// TIA Portal V17 export
// export: Created 2025-03-05T08:01:40.0178288Z, ExportSetting WithDefaults, DisplayName Totally Integrated Automation Portal, DisplayVersion V17 Update 8, DisplayName TIA Portal Openness, DisplayVersion V17 Update 8, DisplayName TIA Portal Version Control Interface, DisplayVersion V17, DisplayName SINAMICS Startdrive Advanced, DisplayVersion V17 SP2, DisplayName SINAMICS Startdrive G110M, G120, G120C, G120D, G120P, G115D, DisplayVersion V17 SP2, DisplayName SINAMICS Startdrive G130, G150, S120, S150, SINAMICS MV, S210, DisplayVersion V17 SP2, DisplayName STEP 7 Professional, DisplayVersion V17 Update 8, DisplayName SINUMERIK ONE STEP 7 Toolbox, DisplayVersion V17 Update 12, DisplayName SINUMERIK 840D sl STEP 7 Toolbox, DisplayVersion V17 Update 12, DisplayName STEP 7 Safety, DisplayVersion V17 Update 6, DisplayName WinCC Advanced, DisplayVersion V17 Update 8
FUNCTION "FC7215_PART_TYPE" : Void   // FC7215, LAD
{ S7_Optimized_Access := 'FALSE' }
AUTHOR : ETXETAR
VERSION : 1.0
// stored: AutoNumber false, IsIECCheckEnabled false, SetENOAutomatically false, UDAEnableTagReadback false
   VAR_TEMP
      PART_TYPE_SCREEN : Int;   // PART TYPE SCREEN
   END_VAR
   VAR CONSTANT
      FC_NUMBER : DInt := 7215;
   END_VAR
   VAR_TEMP   // added for the SCL form of the ladder/FBD networks
      _w1 : Bool;
      _w2 : Bool;
   END_VAR
BEGIN

REGION Network 1: AUTO PART TYPE SELECT
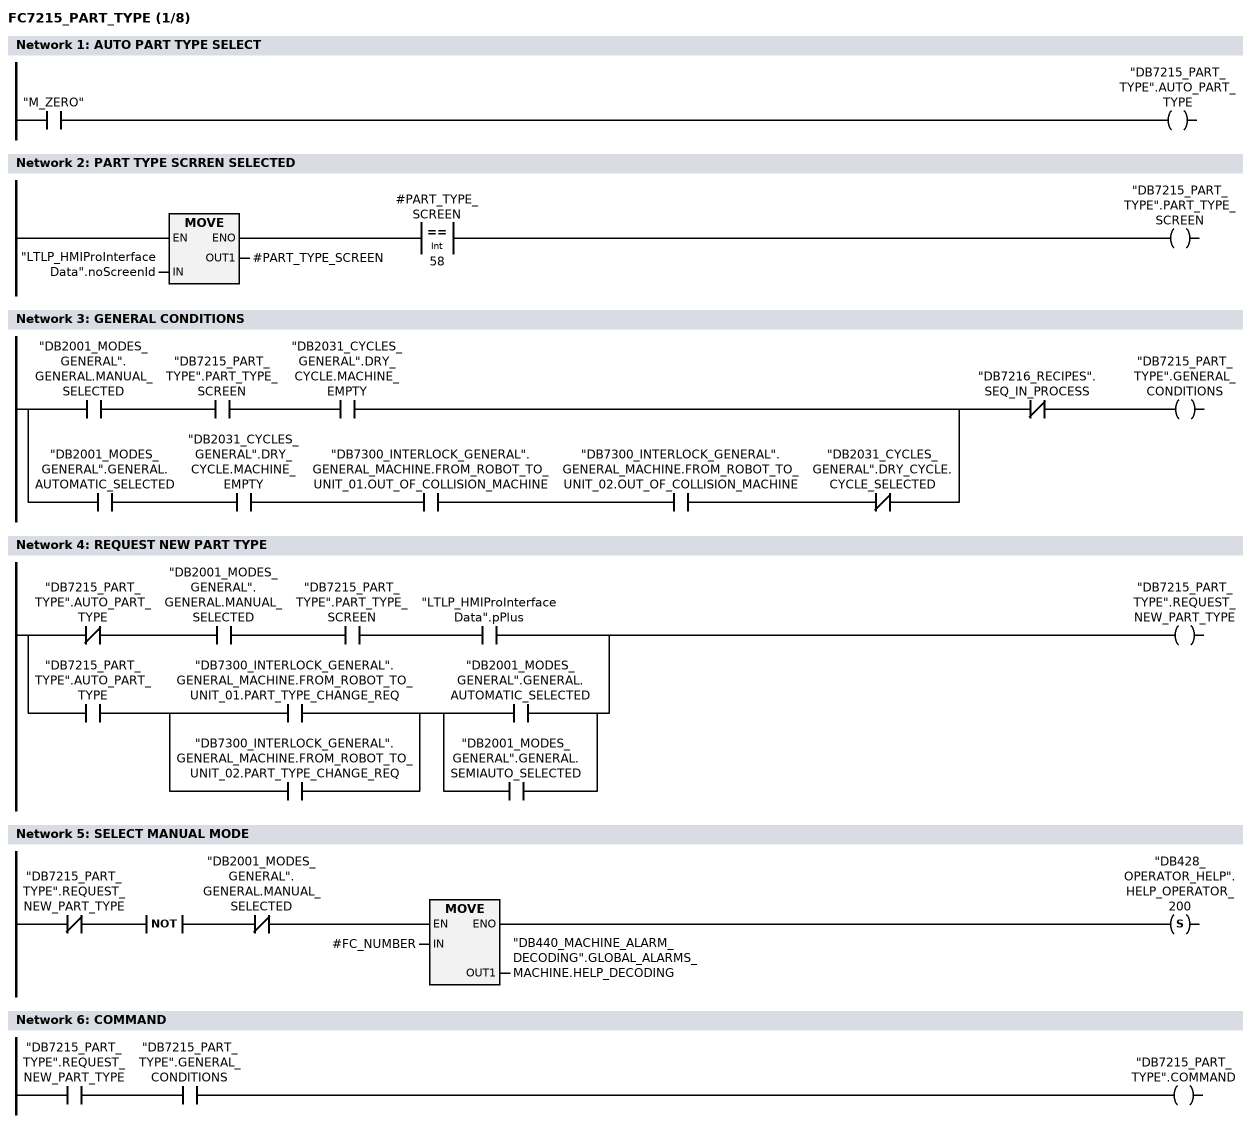
   RUNG wire#powerrail
      Contact( "M_ZERO" )
      Coil( "DB7215_PART_TYPE".AUTO_PART_TYPE )
   END_RUNG
   // the same network as SCL:
   "DB7215_PART_TYPE".AUTO_PART_TYPE := "M_ZERO";
END_REGION

REGION Network 2: PART TYPE SCRREN SELECTED
   RUNG wire#powerrail
      { S7_GenerateENO := "TRUE" } Move(in := "LTLP_HMIProInterfaceData".noScreenId, out1 => #PART_TYPE_SCREEN)
      { S7_Templates := "SrcType := Int" } EQ_Contact(in1 := #PART_TYPE_SCREEN, in2 := 58)
      Coil( "DB7215_PART_TYPE".PART_TYPE_SCREEN )
   END_RUNG
   // the same network as SCL:
   // ENO of a box is taken as its EN; it also drops when the box reports an error
   #PART_TYPE_SCREEN := "LTLP_HMIProInterfaceData".noScreenId;
   "DB7215_PART_TYPE".PART_TYPE_SCREEN := #PART_TYPE_SCREEN = 58;
END_REGION

REGION Network 3: GENERAL CONDITIONS
   RUNG wire#powerrail
      Contact( "DB2001_MODES_GENERAL".GENERAL.MANUAL_SELECTED )
      Contact( "DB7215_PART_TYPE".PART_TYPE_SCREEN )
      Contact( "DB2031_CYCLES_GENERAL".DRY_CYCLE.MACHINE_EMPTY )
      wire#w1
      I_Contact( "DB7216_RECIPES".SEQ_IN_PROCESS )
      Coil( "DB7215_PART_TYPE".GENERAL_CONDITIONS )
   END_RUNG
   RUNG wire#powerrail
      Contact( "DB2001_MODES_GENERAL".GENERAL.AUTOMATIC_SELECTED )
      Contact( "DB2031_CYCLES_GENERAL".DRY_CYCLE.MACHINE_EMPTY )
      Contact( "DB7300_INTERLOCK_GENERAL".GENERAL_MACHINE.FROM_ROBOT_TO_UNIT_01.OUT_OF_COLLISION_MACHINE )
      Contact( "DB7300_INTERLOCK_GENERAL".GENERAL_MACHINE.FROM_ROBOT_TO_UNIT_02.OUT_OF_COLLISION_MACHINE )
      I_Contact( "DB2031_CYCLES_GENERAL".DRY_CYCLE.CYCLE_SELECTED )
   END_RUNG wire#w1
   // the same network as SCL:
   "DB7215_PART_TYPE".GENERAL_CONDITIONS := (("DB2001_MODES_GENERAL".GENERAL.MANUAL_SELECTED AND "DB7215_PART_TYPE".PART_TYPE_SCREEN AND "DB2031_CYCLES_GENERAL".DRY_CYCLE.MACHINE_EMPTY) OR ("DB2001_MODES_GENERAL".GENERAL.AUTOMATIC_SELECTED AND "DB2031_CYCLES_GENERAL".DRY_CYCLE.MACHINE_EMPTY AND "DB7300_INTERLOCK_GENERAL".GENERAL_MACHINE.FROM_ROBOT_TO_UNIT_01.OUT_OF_COLLISION_MACHINE AND "DB7300_INTERLOCK_GENERAL".GENERAL_MACHINE.FROM_ROBOT_TO_UNIT_02.OUT_OF_COLLISION_MACHINE AND NOT "DB2031_CYCLES_GENERAL".DRY_CYCLE.CYCLE_SELECTED)) AND NOT "DB7216_RECIPES".SEQ_IN_PROCESS;
END_REGION

REGION Network 4: REQUEST NEW PART TYPE
   RUNG wire#powerrail
      I_Contact( "DB7215_PART_TYPE".AUTO_PART_TYPE )
      Contact( "DB2001_MODES_GENERAL".GENERAL.MANUAL_SELECTED )
      Contact( "DB7215_PART_TYPE".PART_TYPE_SCREEN )
      Contact( "LTLP_HMIProInterfaceData".pPlus )
      wire#w1
      Coil( "DB7215_PART_TYPE".REQUEST_NEW_PART_TYPE )
   END_RUNG
   RUNG wire#powerrail
      Contact( "DB7215_PART_TYPE".AUTO_PART_TYPE )
      wire#w2
      Contact( "DB7300_INTERLOCK_GENERAL".GENERAL_MACHINE.FROM_ROBOT_TO_UNIT_01.PART_TYPE_CHANGE_REQ )
      wire#w3
      Contact( "DB2001_MODES_GENERAL".GENERAL.AUTOMATIC_SELECTED )
   END_RUNG wire#w1
   RUNG wire#w2
      Contact( "DB7300_INTERLOCK_GENERAL".GENERAL_MACHINE.FROM_ROBOT_TO_UNIT_02.PART_TYPE_CHANGE_REQ )
   END_RUNG wire#w3
   RUNG wire#w3
      Contact( "DB2001_MODES_GENERAL".GENERAL.SEMIAUTO_SELECTED )
   END_RUNG wire#w1
   // the same network as SCL:
   "DB7215_PART_TYPE".REQUEST_NEW_PART_TYPE := (NOT "DB7215_PART_TYPE".AUTO_PART_TYPE AND "DB2001_MODES_GENERAL".GENERAL.MANUAL_SELECTED AND "DB7215_PART_TYPE".PART_TYPE_SCREEN AND "LTLP_HMIProInterfaceData".pPlus) OR ("DB7215_PART_TYPE".AUTO_PART_TYPE AND ("DB7300_INTERLOCK_GENERAL".GENERAL_MACHINE.FROM_ROBOT_TO_UNIT_01.PART_TYPE_CHANGE_REQ OR "DB7300_INTERLOCK_GENERAL".GENERAL_MACHINE.FROM_ROBOT_TO_UNIT_02.PART_TYPE_CHANGE_REQ) AND ("DB2001_MODES_GENERAL".GENERAL.AUTOMATIC_SELECTED OR "DB2001_MODES_GENERAL".GENERAL.SEMIAUTO_SELECTED));
END_REGION

REGION Network 5: SELECT MANUAL MODE
   RUNG wire#powerrail
      I_Contact( "DB7215_PART_TYPE".REQUEST_NEW_PART_TYPE )
      Not()
      I_Contact( "DB2001_MODES_GENERAL".GENERAL.MANUAL_SELECTED )
      { S7_GenerateENO := "TRUE" } Move(in := #FC_NUMBER, out1 => "DB440_MACHINE_ALARM_DECODING".GLOBAL_ALARMS_MACHINE.HELP_DECODING)
      S_Coil( "DB428_OPERATOR_HELP".HELP_OPERATOR_200 )
   END_RUNG
   // the same network as SCL:
   // ENO of a box is taken as its EN; it also drops when the box reports an error
   IF NOT (NOT "DB7215_PART_TYPE".REQUEST_NEW_PART_TYPE) AND NOT "DB2001_MODES_GENERAL".GENERAL.MANUAL_SELECTED THEN
       "DB440_MACHINE_ALARM_DECODING".GLOBAL_ALARMS_MACHINE.HELP_DECODING := #FC_NUMBER;
       "DB428_OPERATOR_HELP".HELP_OPERATOR_200 := TRUE;
   END_IF;
END_REGION

REGION Network 6: COMMAND
   RUNG wire#powerrail
      Contact( "DB7215_PART_TYPE".REQUEST_NEW_PART_TYPE )
      Contact( "DB7215_PART_TYPE".GENERAL_CONDITIONS )
      Coil( "DB7215_PART_TYPE".COMMAND )
   END_RUNG
   // the same network as SCL:
   "DB7215_PART_TYPE".COMMAND := "DB7215_PART_TYPE".REQUEST_NEW_PART_TYPE AND "DB7215_PART_TYPE".GENERAL_CONDITIONS;
END_REGION

REGION Network 7: COMMAND
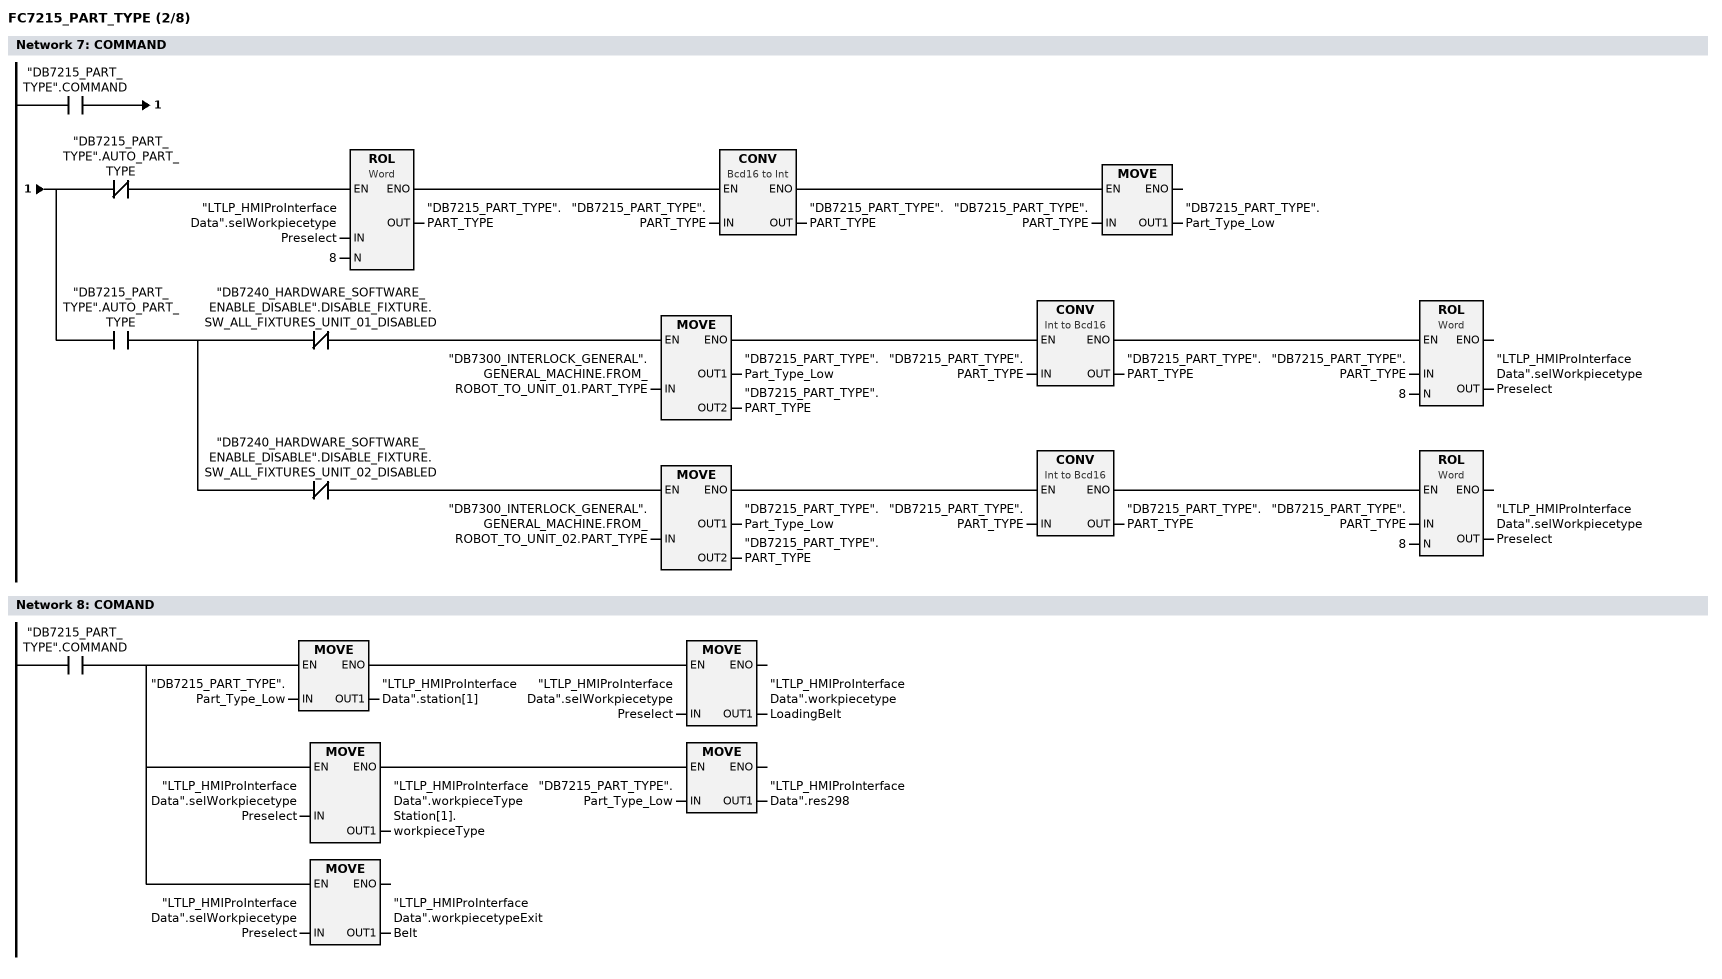
   IF "DB7215_PART_TYPE".COMMAND AND NOT "DB7215_PART_TYPE".AUTO_PART_TYPE THEN
       "DB7215_PART_TYPE".PART_TYPE := ROL(IN := "LTLP_HMIProInterfaceData".selWorkpiecetypePreselect, N := 8);
       "DB7215_PART_TYPE".PART_TYPE := BCD16_TO_INT("DB7215_PART_TYPE".PART_TYPE);
       "DB7215_PART_TYPE".Part_Type_Low := "DB7215_PART_TYPE".PART_TYPE;
   END_IF;
   #_w1 := "DB7215_PART_TYPE".COMMAND AND "DB7215_PART_TYPE".AUTO_PART_TYPE;
   IF #_w1 AND NOT "DB7240_HARDWARE_SOFTWARE_ENABLE_DISABLE".DISABLE_FIXTURE.SW_ALL_FIXTURES_UNIT_01_DISABLED THEN
       "DB7215_PART_TYPE".Part_Type_Low := "DB7300_INTERLOCK_GENERAL".GENERAL_MACHINE.FROM_ROBOT_TO_UNIT_01.PART_TYPE;
       "DB7215_PART_TYPE".PART_TYPE := "DB7300_INTERLOCK_GENERAL".GENERAL_MACHINE.FROM_ROBOT_TO_UNIT_01.PART_TYPE;
       "DB7215_PART_TYPE".PART_TYPE := INT_TO_BCD16("DB7215_PART_TYPE".PART_TYPE);
       "LTLP_HMIProInterfaceData".selWorkpiecetypePreselect := ROL(IN := "DB7215_PART_TYPE".PART_TYPE, N := 8);
   END_IF;
   IF #_w1 AND NOT "DB7240_HARDWARE_SOFTWARE_ENABLE_DISABLE".DISABLE_FIXTURE.SW_ALL_FIXTURES_UNIT_02_DISABLED THEN
       "DB7215_PART_TYPE".Part_Type_Low := "DB7300_INTERLOCK_GENERAL".GENERAL_MACHINE.FROM_ROBOT_TO_UNIT_02.PART_TYPE;
       "DB7215_PART_TYPE".PART_TYPE := "DB7300_INTERLOCK_GENERAL".GENERAL_MACHINE.FROM_ROBOT_TO_UNIT_02.PART_TYPE;
       "DB7215_PART_TYPE".PART_TYPE := INT_TO_BCD16("DB7215_PART_TYPE".PART_TYPE);
       "LTLP_HMIProInterfaceData".selWorkpiecetypePreselect := ROL(IN := "DB7215_PART_TYPE".PART_TYPE, N := 8);
   END_IF;
END_REGION

REGION Network 8: COMAND
   RUNG wire#powerrail
      Contact( "DB7215_PART_TYPE".COMMAND )
      wire#w1
      { S7_GenerateENO := "TRUE" } Move(in := "DB7215_PART_TYPE".Part_Type_Low, out1 => "LTLP_HMIProInterfaceData".station[1])
      { S7_GenerateENO := "TRUE" } Move(in := "LTLP_HMIProInterfaceData".selWorkpiecetypePreselect, out1 => "LTLP_HMIProInterfaceData".workpiecetypeLoadingBelt)
   END_RUNG
   RUNG wire#w1
      { S7_GenerateENO := "TRUE" } Move(in := "LTLP_HMIProInterfaceData".selWorkpiecetypePreselect, out1 => "LTLP_HMIProInterfaceData".workpieceTypeStation[1].workpieceType)
      { S7_GenerateENO := "TRUE" } Move(in := "DB7215_PART_TYPE".Part_Type_Low, out1 => "LTLP_HMIProInterfaceData".res298)
   END_RUNG
   RUNG wire#w1
      { S7_GenerateENO := "TRUE" } Move(in := "LTLP_HMIProInterfaceData".selWorkpiecetypePreselect, out1 => "LTLP_HMIProInterfaceData".workpiecetypeExitBelt)
   END_RUNG
   // the same network as SCL:
   // ENO of a box is taken as its EN; it also drops when the box reports an error
   IF "DB7215_PART_TYPE".COMMAND THEN
       "LTLP_HMIProInterfaceData".station[1] := "DB7215_PART_TYPE".Part_Type_Low;
       "LTLP_HMIProInterfaceData".workpiecetypeLoadingBelt := "LTLP_HMIProInterfaceData".selWorkpiecetypePreselect;
       "LTLP_HMIProInterfaceData".workpieceTypeStation[1].workpieceType := "LTLP_HMIProInterfaceData".selWorkpiecetypePreselect;
       "LTLP_HMIProInterfaceData".res298 := "DB7215_PART_TYPE".Part_Type_Low;
       "LTLP_HMIProInterfaceData".workpiecetypeExitBelt := "LTLP_HMIProInterfaceData".selWorkpiecetypePreselect;
   END_IF;
END_REGION

REGION Network 9: PART TYPE SELECTED 1 - 8
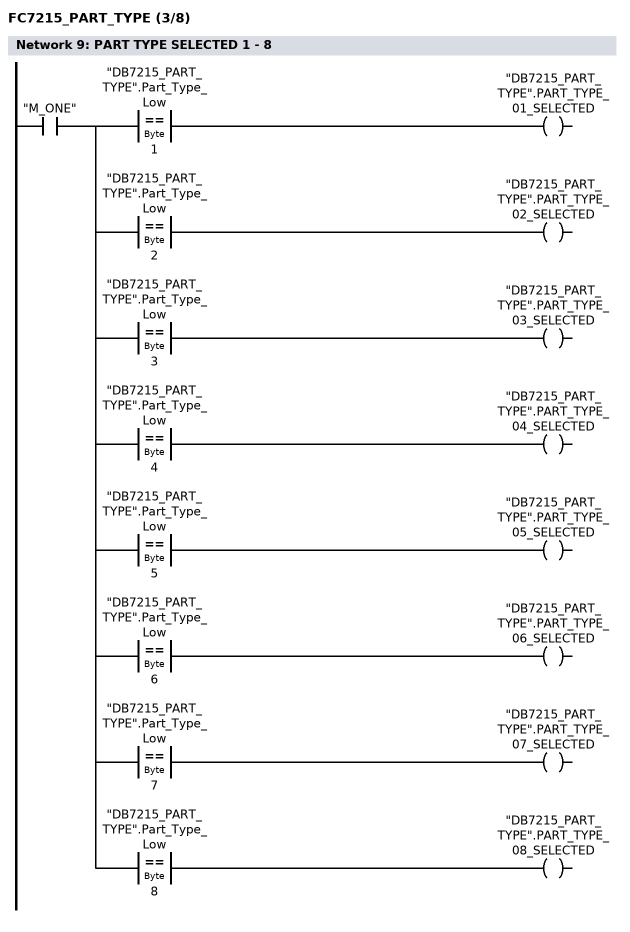
   RUNG wire#powerrail
      Contact( "M_ONE" )
      wire#w1
      { S7_Templates := "SrcType := Byte" } EQ_Contact(in1 := "DB7215_PART_TYPE".Part_Type_Low, in2 := 1)
      Coil( "DB7215_PART_TYPE".PART_TYPE_01_SELECTED )
   END_RUNG
   RUNG wire#w1
      { S7_Templates := "SrcType := Byte" } EQ_Contact(in1 := "DB7215_PART_TYPE".Part_Type_Low, in2 := 2)
      Coil( "DB7215_PART_TYPE".PART_TYPE_02_SELECTED )
   END_RUNG
   RUNG wire#w1
      { S7_Templates := "SrcType := Byte" } EQ_Contact(in1 := "DB7215_PART_TYPE".Part_Type_Low, in2 := 3)
      Coil( "DB7215_PART_TYPE".PART_TYPE_03_SELECTED )
   END_RUNG
   RUNG wire#w1
      { S7_Templates := "SrcType := Byte" } EQ_Contact(in1 := "DB7215_PART_TYPE".Part_Type_Low, in2 := 4)
      Coil( "DB7215_PART_TYPE".PART_TYPE_04_SELECTED )
   END_RUNG
   RUNG wire#w1
      { S7_Templates := "SrcType := Byte" } EQ_Contact(in1 := "DB7215_PART_TYPE".Part_Type_Low, in2 := 5)
      Coil( "DB7215_PART_TYPE".PART_TYPE_05_SELECTED )
   END_RUNG
   RUNG wire#w1
      { S7_Templates := "SrcType := Byte" } EQ_Contact(in1 := "DB7215_PART_TYPE".Part_Type_Low, in2 := 6)
      Coil( "DB7215_PART_TYPE".PART_TYPE_06_SELECTED )
   END_RUNG
   RUNG wire#w1
      { S7_Templates := "SrcType := Byte" } EQ_Contact(in1 := "DB7215_PART_TYPE".Part_Type_Low, in2 := 7)
      Coil( "DB7215_PART_TYPE".PART_TYPE_07_SELECTED )
   END_RUNG
   RUNG wire#w1
      { S7_Templates := "SrcType := Byte" } EQ_Contact(in1 := "DB7215_PART_TYPE".Part_Type_Low, in2 := 8)
      Coil( "DB7215_PART_TYPE".PART_TYPE_08_SELECTED )
   END_RUNG
   // the same network as SCL:
   "DB7215_PART_TYPE".PART_TYPE_01_SELECTED := "M_ONE" AND ("DB7215_PART_TYPE".Part_Type_Low = 1);
   "DB7215_PART_TYPE".PART_TYPE_02_SELECTED := "M_ONE" AND ("DB7215_PART_TYPE".Part_Type_Low = 2);
   "DB7215_PART_TYPE".PART_TYPE_03_SELECTED := "M_ONE" AND ("DB7215_PART_TYPE".Part_Type_Low = 3);
   "DB7215_PART_TYPE".PART_TYPE_04_SELECTED := "M_ONE" AND ("DB7215_PART_TYPE".Part_Type_Low = 4);
   "DB7215_PART_TYPE".PART_TYPE_05_SELECTED := "M_ONE" AND ("DB7215_PART_TYPE".Part_Type_Low = 5);
   "DB7215_PART_TYPE".PART_TYPE_06_SELECTED := "M_ONE" AND ("DB7215_PART_TYPE".Part_Type_Low = 6);
   "DB7215_PART_TYPE".PART_TYPE_07_SELECTED := "M_ONE" AND ("DB7215_PART_TYPE".Part_Type_Low = 7);
   "DB7215_PART_TYPE".PART_TYPE_08_SELECTED := "M_ONE" AND ("DB7215_PART_TYPE".Part_Type_Low = 8);
END_REGION

REGION Network 10: PART TYPE SELECTED 9 - 16
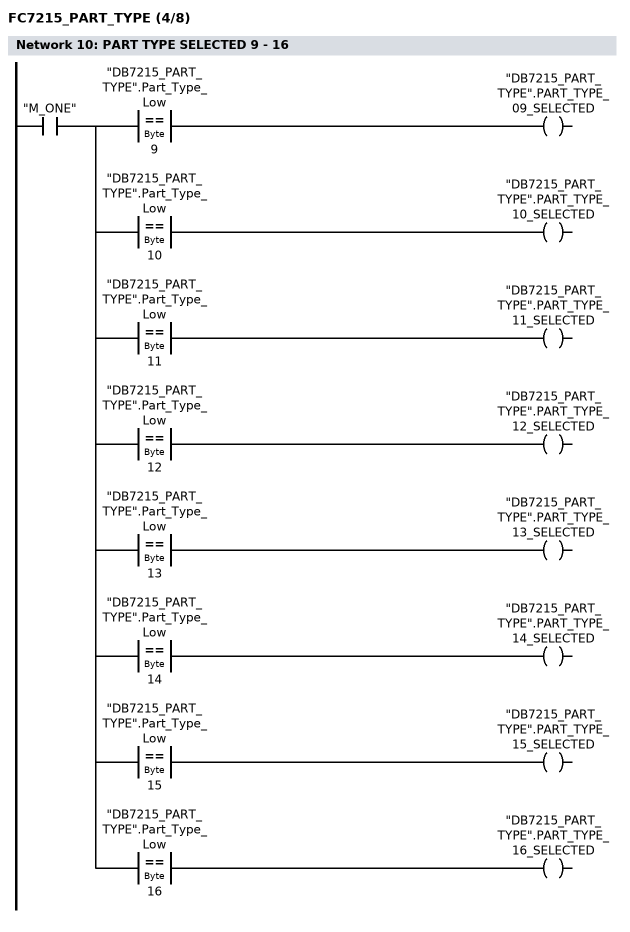
   RUNG wire#powerrail
      Contact( "M_ONE" )
      wire#w1
      { S7_Templates := "SrcType := Byte" } EQ_Contact(in1 := "DB7215_PART_TYPE".Part_Type_Low, in2 := 9)
      Coil( "DB7215_PART_TYPE".PART_TYPE_09_SELECTED )
   END_RUNG
   RUNG wire#w1
      { S7_Templates := "SrcType := Byte" } EQ_Contact(in1 := "DB7215_PART_TYPE".Part_Type_Low, in2 := 10)
      Coil( "DB7215_PART_TYPE".PART_TYPE_10_SELECTED )
   END_RUNG
   RUNG wire#w1
      { S7_Templates := "SrcType := Byte" } EQ_Contact(in1 := "DB7215_PART_TYPE".Part_Type_Low, in2 := 11)
      Coil( "DB7215_PART_TYPE".PART_TYPE_11_SELECTED )
   END_RUNG
   RUNG wire#w1
      { S7_Templates := "SrcType := Byte" } EQ_Contact(in1 := "DB7215_PART_TYPE".Part_Type_Low, in2 := 12)
      Coil( "DB7215_PART_TYPE".PART_TYPE_12_SELECTED )
   END_RUNG
   RUNG wire#w1
      { S7_Templates := "SrcType := Byte" } EQ_Contact(in1 := "DB7215_PART_TYPE".Part_Type_Low, in2 := 13)
      Coil( "DB7215_PART_TYPE".PART_TYPE_13_SELECTED )
   END_RUNG
   RUNG wire#w1
      { S7_Templates := "SrcType := Byte" } EQ_Contact(in1 := "DB7215_PART_TYPE".Part_Type_Low, in2 := 14)
      Coil( "DB7215_PART_TYPE".PART_TYPE_14_SELECTED )
   END_RUNG
   RUNG wire#w1
      { S7_Templates := "SrcType := Byte" } EQ_Contact(in1 := "DB7215_PART_TYPE".Part_Type_Low, in2 := 15)
      Coil( "DB7215_PART_TYPE".PART_TYPE_15_SELECTED )
   END_RUNG
   RUNG wire#w1
      { S7_Templates := "SrcType := Byte" } EQ_Contact(in1 := "DB7215_PART_TYPE".Part_Type_Low, in2 := 16)
      Coil( "DB7215_PART_TYPE".PART_TYPE_16_SELECTED )
   END_RUNG
   // the same network as SCL:
   "DB7215_PART_TYPE".PART_TYPE_09_SELECTED := "M_ONE" AND ("DB7215_PART_TYPE".Part_Type_Low = 9);
   "DB7215_PART_TYPE".PART_TYPE_10_SELECTED := "M_ONE" AND ("DB7215_PART_TYPE".Part_Type_Low = 10);
   "DB7215_PART_TYPE".PART_TYPE_11_SELECTED := "M_ONE" AND ("DB7215_PART_TYPE".Part_Type_Low = 11);
   "DB7215_PART_TYPE".PART_TYPE_12_SELECTED := "M_ONE" AND ("DB7215_PART_TYPE".Part_Type_Low = 12);
   "DB7215_PART_TYPE".PART_TYPE_13_SELECTED := "M_ONE" AND ("DB7215_PART_TYPE".Part_Type_Low = 13);
   "DB7215_PART_TYPE".PART_TYPE_14_SELECTED := "M_ONE" AND ("DB7215_PART_TYPE".Part_Type_Low = 14);
   "DB7215_PART_TYPE".PART_TYPE_15_SELECTED := "M_ONE" AND ("DB7215_PART_TYPE".Part_Type_Low = 15);
   "DB7215_PART_TYPE".PART_TYPE_16_SELECTED := "M_ONE" AND ("DB7215_PART_TYPE".Part_Type_Low = 16);
END_REGION

REGION Network 11: PART TYPE SELECTED 17 - 24
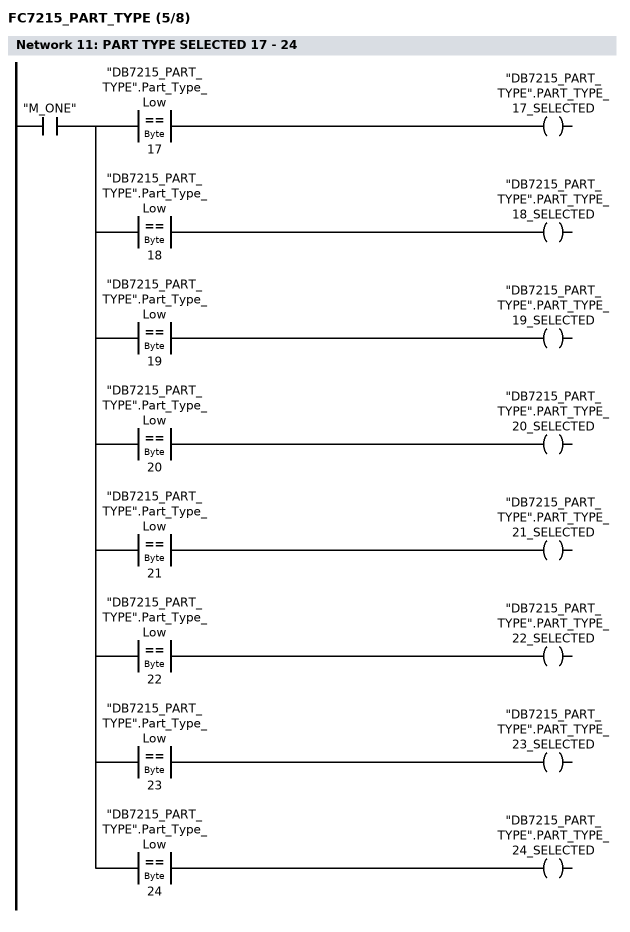
   RUNG wire#powerrail
      Contact( "M_ONE" )
      wire#w1
      { S7_Templates := "SrcType := Byte" } EQ_Contact(in1 := "DB7215_PART_TYPE".Part_Type_Low, in2 := 17)
      Coil( "DB7215_PART_TYPE".PART_TYPE_17_SELECTED )
   END_RUNG
   RUNG wire#w1
      { S7_Templates := "SrcType := Byte" } EQ_Contact(in1 := "DB7215_PART_TYPE".Part_Type_Low, in2 := 18)
      Coil( "DB7215_PART_TYPE".PART_TYPE_18_SELECTED )
   END_RUNG
   RUNG wire#w1
      { S7_Templates := "SrcType := Byte" } EQ_Contact(in1 := "DB7215_PART_TYPE".Part_Type_Low, in2 := 19)
      Coil( "DB7215_PART_TYPE".PART_TYPE_19_SELECTED )
   END_RUNG
   RUNG wire#w1
      { S7_Templates := "SrcType := Byte" } EQ_Contact(in1 := "DB7215_PART_TYPE".Part_Type_Low, in2 := 20)
      Coil( "DB7215_PART_TYPE".PART_TYPE_20_SELECTED )
   END_RUNG
   RUNG wire#w1
      { S7_Templates := "SrcType := Byte" } EQ_Contact(in1 := "DB7215_PART_TYPE".Part_Type_Low, in2 := 21)
      Coil( "DB7215_PART_TYPE".PART_TYPE_21_SELECTED )
   END_RUNG
   RUNG wire#w1
      { S7_Templates := "SrcType := Byte" } EQ_Contact(in1 := "DB7215_PART_TYPE".Part_Type_Low, in2 := 22)
      Coil( "DB7215_PART_TYPE".PART_TYPE_22_SELECTED )
   END_RUNG
   RUNG wire#w1
      { S7_Templates := "SrcType := Byte" } EQ_Contact(in1 := "DB7215_PART_TYPE".Part_Type_Low, in2 := 23)
      Coil( "DB7215_PART_TYPE".PART_TYPE_23_SELECTED )
   END_RUNG
   RUNG wire#w1
      { S7_Templates := "SrcType := Byte" } EQ_Contact(in1 := "DB7215_PART_TYPE".Part_Type_Low, in2 := 24)
      Coil( "DB7215_PART_TYPE".PART_TYPE_24_SELECTED )
   END_RUNG
   // the same network as SCL:
   "DB7215_PART_TYPE".PART_TYPE_17_SELECTED := "M_ONE" AND ("DB7215_PART_TYPE".Part_Type_Low = 17);
   "DB7215_PART_TYPE".PART_TYPE_18_SELECTED := "M_ONE" AND ("DB7215_PART_TYPE".Part_Type_Low = 18);
   "DB7215_PART_TYPE".PART_TYPE_19_SELECTED := "M_ONE" AND ("DB7215_PART_TYPE".Part_Type_Low = 19);
   "DB7215_PART_TYPE".PART_TYPE_20_SELECTED := "M_ONE" AND ("DB7215_PART_TYPE".Part_Type_Low = 20);
   "DB7215_PART_TYPE".PART_TYPE_21_SELECTED := "M_ONE" AND ("DB7215_PART_TYPE".Part_Type_Low = 21);
   "DB7215_PART_TYPE".PART_TYPE_22_SELECTED := "M_ONE" AND ("DB7215_PART_TYPE".Part_Type_Low = 22);
   "DB7215_PART_TYPE".PART_TYPE_23_SELECTED := "M_ONE" AND ("DB7215_PART_TYPE".Part_Type_Low = 23);
   "DB7215_PART_TYPE".PART_TYPE_24_SELECTED := "M_ONE" AND ("DB7215_PART_TYPE".Part_Type_Low = 24);
END_REGION

REGION Network 12: PART TYPE SELECTED 25 - 32
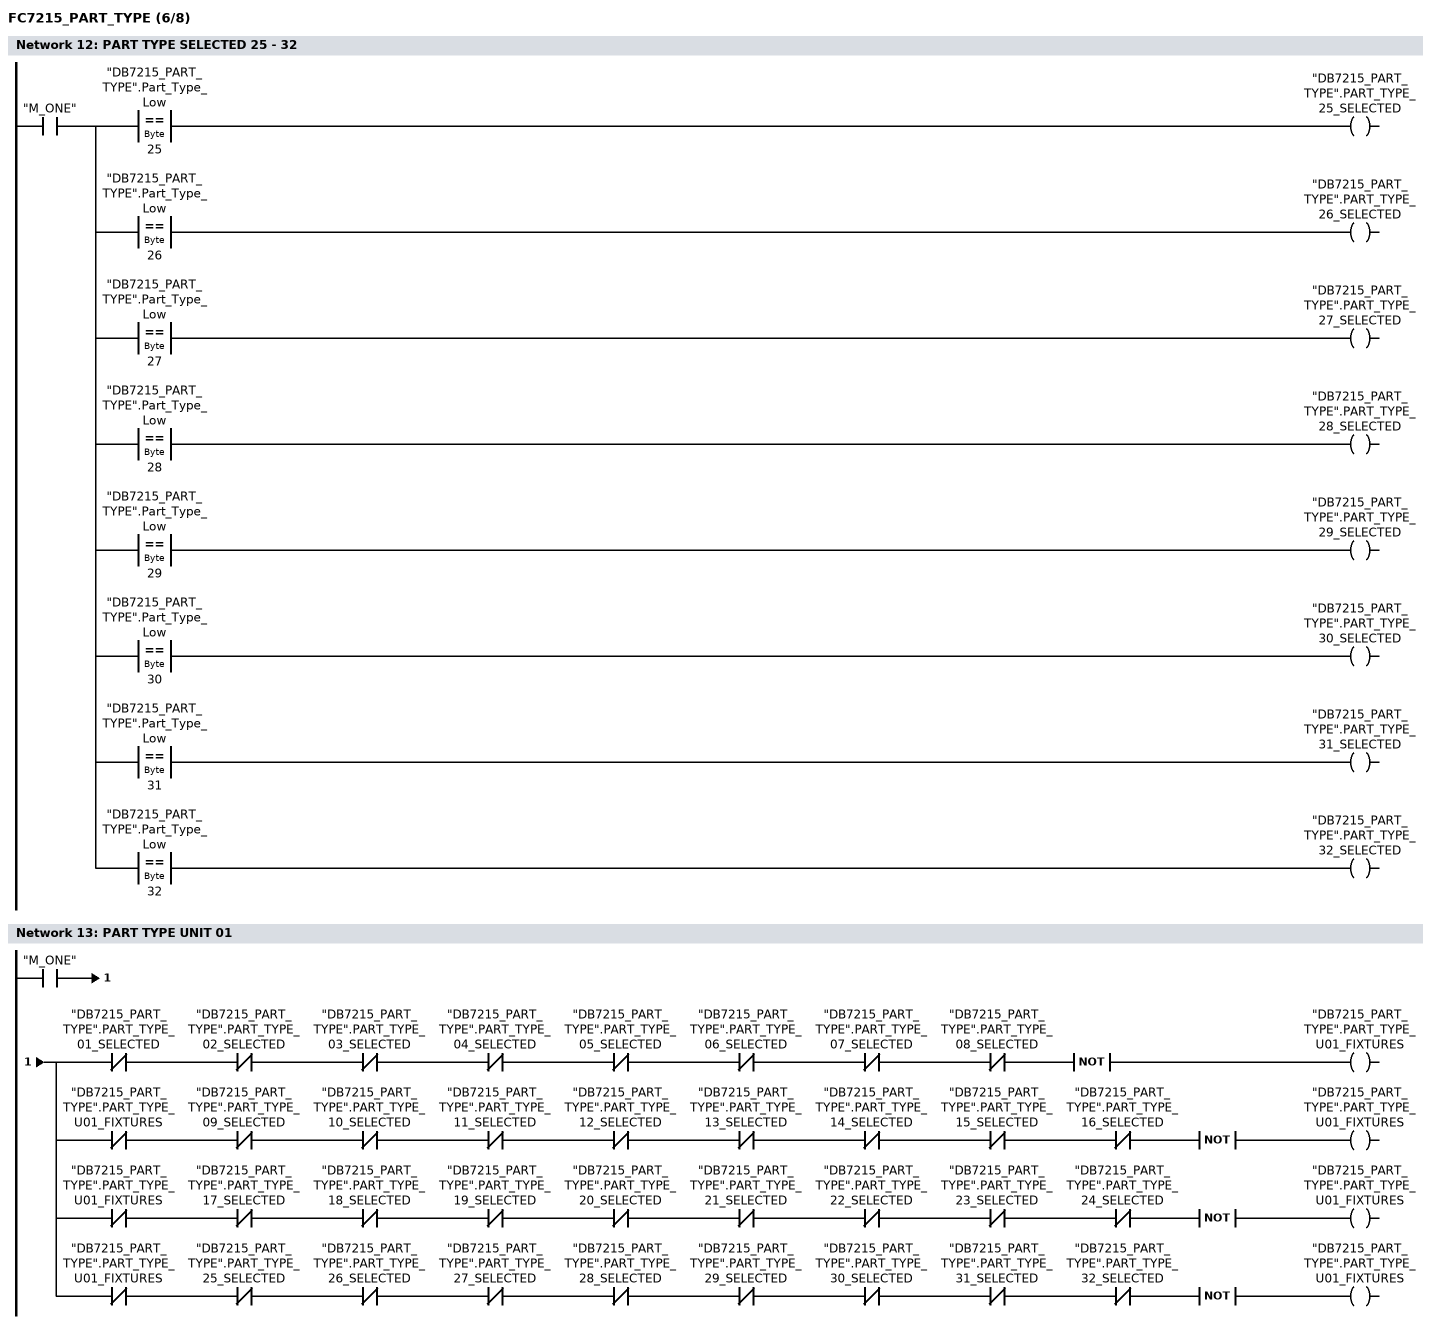
   RUNG wire#powerrail
      Contact( "M_ONE" )
      wire#w1
      { S7_Templates := "SrcType := Byte" } EQ_Contact(in1 := "DB7215_PART_TYPE".Part_Type_Low, in2 := 25)
      Coil( "DB7215_PART_TYPE".PART_TYPE_25_SELECTED )
   END_RUNG
   RUNG wire#w1
      { S7_Templates := "SrcType := Byte" } EQ_Contact(in1 := "DB7215_PART_TYPE".Part_Type_Low, in2 := 26)
      Coil( "DB7215_PART_TYPE".PART_TYPE_26_SELECTED )
   END_RUNG
   RUNG wire#w1
      { S7_Templates := "SrcType := Byte" } EQ_Contact(in1 := "DB7215_PART_TYPE".Part_Type_Low, in2 := 27)
      Coil( "DB7215_PART_TYPE".PART_TYPE_27_SELECTED )
   END_RUNG
   RUNG wire#w1
      { S7_Templates := "SrcType := Byte" } EQ_Contact(in1 := "DB7215_PART_TYPE".Part_Type_Low, in2 := 28)
      Coil( "DB7215_PART_TYPE".PART_TYPE_28_SELECTED )
   END_RUNG
   RUNG wire#w1
      { S7_Templates := "SrcType := Byte" } EQ_Contact(in1 := "DB7215_PART_TYPE".Part_Type_Low, in2 := 29)
      Coil( "DB7215_PART_TYPE".PART_TYPE_29_SELECTED )
   END_RUNG
   RUNG wire#w1
      { S7_Templates := "SrcType := Byte" } EQ_Contact(in1 := "DB7215_PART_TYPE".Part_Type_Low, in2 := 30)
      Coil( "DB7215_PART_TYPE".PART_TYPE_30_SELECTED )
   END_RUNG
   RUNG wire#w1
      { S7_Templates := "SrcType := Byte" } EQ_Contact(in1 := "DB7215_PART_TYPE".Part_Type_Low, in2 := 31)
      Coil( "DB7215_PART_TYPE".PART_TYPE_31_SELECTED )
   END_RUNG
   RUNG wire#w1
      { S7_Templates := "SrcType := Byte" } EQ_Contact(in1 := "DB7215_PART_TYPE".Part_Type_Low, in2 := 32)
      Coil( "DB7215_PART_TYPE".PART_TYPE_32_SELECTED )
   END_RUNG
   // the same network as SCL:
   "DB7215_PART_TYPE".PART_TYPE_25_SELECTED := "M_ONE" AND ("DB7215_PART_TYPE".Part_Type_Low = 25);
   "DB7215_PART_TYPE".PART_TYPE_26_SELECTED := "M_ONE" AND ("DB7215_PART_TYPE".Part_Type_Low = 26);
   "DB7215_PART_TYPE".PART_TYPE_27_SELECTED := "M_ONE" AND ("DB7215_PART_TYPE".Part_Type_Low = 27);
   "DB7215_PART_TYPE".PART_TYPE_28_SELECTED := "M_ONE" AND ("DB7215_PART_TYPE".Part_Type_Low = 28);
   "DB7215_PART_TYPE".PART_TYPE_29_SELECTED := "M_ONE" AND ("DB7215_PART_TYPE".Part_Type_Low = 29);
   "DB7215_PART_TYPE".PART_TYPE_30_SELECTED := "M_ONE" AND ("DB7215_PART_TYPE".Part_Type_Low = 30);
   "DB7215_PART_TYPE".PART_TYPE_31_SELECTED := "M_ONE" AND ("DB7215_PART_TYPE".Part_Type_Low = 31);
   "DB7215_PART_TYPE".PART_TYPE_32_SELECTED := "M_ONE" AND ("DB7215_PART_TYPE".Part_Type_Low = 32);
END_REGION

REGION Network 13: PART TYPE UNIT 01
   RUNG wire#powerrail
      Contact( "M_ONE" )
      wire#w1
      I_Contact( "DB7215_PART_TYPE".PART_TYPE_01_SELECTED )
      I_Contact( "DB7215_PART_TYPE".PART_TYPE_02_SELECTED )
      I_Contact( "DB7215_PART_TYPE".PART_TYPE_03_SELECTED )
      I_Contact( "DB7215_PART_TYPE".PART_TYPE_04_SELECTED )
      I_Contact( "DB7215_PART_TYPE".PART_TYPE_05_SELECTED )
      I_Contact( "DB7215_PART_TYPE".PART_TYPE_06_SELECTED )
      I_Contact( "DB7215_PART_TYPE".PART_TYPE_07_SELECTED )
      I_Contact( "DB7215_PART_TYPE".PART_TYPE_08_SELECTED )
      Not()
      Coil( "DB7215_PART_TYPE".PART_TYPE_U01_FIXTURES )
   END_RUNG
   RUNG wire#w1
      I_Contact( "DB7215_PART_TYPE".PART_TYPE_U01_FIXTURES )
      I_Contact( "DB7215_PART_TYPE".PART_TYPE_09_SELECTED )
      I_Contact( "DB7215_PART_TYPE".PART_TYPE_10_SELECTED )
      I_Contact( "DB7215_PART_TYPE".PART_TYPE_11_SELECTED )
      I_Contact( "DB7215_PART_TYPE".PART_TYPE_12_SELECTED )
      I_Contact( "DB7215_PART_TYPE".PART_TYPE_13_SELECTED )
      I_Contact( "DB7215_PART_TYPE".PART_TYPE_14_SELECTED )
      I_Contact( "DB7215_PART_TYPE".PART_TYPE_15_SELECTED )
      I_Contact( "DB7215_PART_TYPE".PART_TYPE_16_SELECTED )
      Not()
      Coil( "DB7215_PART_TYPE".PART_TYPE_U01_FIXTURES )
   END_RUNG
   RUNG wire#w1
      I_Contact( "DB7215_PART_TYPE".PART_TYPE_U01_FIXTURES )
      I_Contact( "DB7215_PART_TYPE".PART_TYPE_17_SELECTED )
      I_Contact( "DB7215_PART_TYPE".PART_TYPE_18_SELECTED )
      I_Contact( "DB7215_PART_TYPE".PART_TYPE_19_SELECTED )
      I_Contact( "DB7215_PART_TYPE".PART_TYPE_20_SELECTED )
      I_Contact( "DB7215_PART_TYPE".PART_TYPE_21_SELECTED )
      I_Contact( "DB7215_PART_TYPE".PART_TYPE_22_SELECTED )
      I_Contact( "DB7215_PART_TYPE".PART_TYPE_23_SELECTED )
      I_Contact( "DB7215_PART_TYPE".PART_TYPE_24_SELECTED )
      Not()
      Coil( "DB7215_PART_TYPE".PART_TYPE_U01_FIXTURES )
   END_RUNG
   RUNG wire#w1
      I_Contact( "DB7215_PART_TYPE".PART_TYPE_U01_FIXTURES )
      I_Contact( "DB7215_PART_TYPE".PART_TYPE_25_SELECTED )
      I_Contact( "DB7215_PART_TYPE".PART_TYPE_26_SELECTED )
      I_Contact( "DB7215_PART_TYPE".PART_TYPE_27_SELECTED )
      I_Contact( "DB7215_PART_TYPE".PART_TYPE_28_SELECTED )
      I_Contact( "DB7215_PART_TYPE".PART_TYPE_29_SELECTED )
      I_Contact( "DB7215_PART_TYPE".PART_TYPE_30_SELECTED )
      I_Contact( "DB7215_PART_TYPE".PART_TYPE_31_SELECTED )
      I_Contact( "DB7215_PART_TYPE".PART_TYPE_32_SELECTED )
      Not()
      Coil( "DB7215_PART_TYPE".PART_TYPE_U01_FIXTURES )
   END_RUNG
   // the same network as SCL:
   "DB7215_PART_TYPE".PART_TYPE_U01_FIXTURES := NOT ("M_ONE" AND NOT "DB7215_PART_TYPE".PART_TYPE_01_SELECTED AND NOT "DB7215_PART_TYPE".PART_TYPE_02_SELECTED AND NOT "DB7215_PART_TYPE".PART_TYPE_03_SELECTED AND NOT "DB7215_PART_TYPE".PART_TYPE_04_SELECTED AND NOT "DB7215_PART_TYPE".PART_TYPE_05_SELECTED AND NOT "DB7215_PART_TYPE".PART_TYPE_06_SELECTED AND NOT "DB7215_PART_TYPE".PART_TYPE_07_SELECTED AND NOT "DB7215_PART_TYPE".PART_TYPE_08_SELECTED);
   "DB7215_PART_TYPE".PART_TYPE_U01_FIXTURES := NOT ("M_ONE" AND NOT "DB7215_PART_TYPE".PART_TYPE_U01_FIXTURES AND NOT "DB7215_PART_TYPE".PART_TYPE_09_SELECTED AND NOT "DB7215_PART_TYPE".PART_TYPE_10_SELECTED AND NOT "DB7215_PART_TYPE".PART_TYPE_11_SELECTED AND NOT "DB7215_PART_TYPE".PART_TYPE_12_SELECTED AND NOT "DB7215_PART_TYPE".PART_TYPE_13_SELECTED AND NOT "DB7215_PART_TYPE".PART_TYPE_14_SELECTED AND NOT "DB7215_PART_TYPE".PART_TYPE_15_SELECTED AND NOT "DB7215_PART_TYPE".PART_TYPE_16_SELECTED);
   "DB7215_PART_TYPE".PART_TYPE_U01_FIXTURES := NOT ("M_ONE" AND NOT "DB7215_PART_TYPE".PART_TYPE_U01_FIXTURES AND NOT "DB7215_PART_TYPE".PART_TYPE_17_SELECTED AND NOT "DB7215_PART_TYPE".PART_TYPE_18_SELECTED AND NOT "DB7215_PART_TYPE".PART_TYPE_19_SELECTED AND NOT "DB7215_PART_TYPE".PART_TYPE_20_SELECTED AND NOT "DB7215_PART_TYPE".PART_TYPE_21_SELECTED AND NOT "DB7215_PART_TYPE".PART_TYPE_22_SELECTED AND NOT "DB7215_PART_TYPE".PART_TYPE_23_SELECTED AND NOT "DB7215_PART_TYPE".PART_TYPE_24_SELECTED);
   "DB7215_PART_TYPE".PART_TYPE_U01_FIXTURES := NOT ("M_ONE" AND NOT "DB7215_PART_TYPE".PART_TYPE_U01_FIXTURES AND NOT "DB7215_PART_TYPE".PART_TYPE_25_SELECTED AND NOT "DB7215_PART_TYPE".PART_TYPE_26_SELECTED AND NOT "DB7215_PART_TYPE".PART_TYPE_27_SELECTED AND NOT "DB7215_PART_TYPE".PART_TYPE_28_SELECTED AND NOT "DB7215_PART_TYPE".PART_TYPE_29_SELECTED AND NOT "DB7215_PART_TYPE".PART_TYPE_30_SELECTED AND NOT "DB7215_PART_TYPE".PART_TYPE_31_SELECTED AND NOT "DB7215_PART_TYPE".PART_TYPE_32_SELECTED);
END_REGION

REGION Network 14: PART TYPE UNIT 02
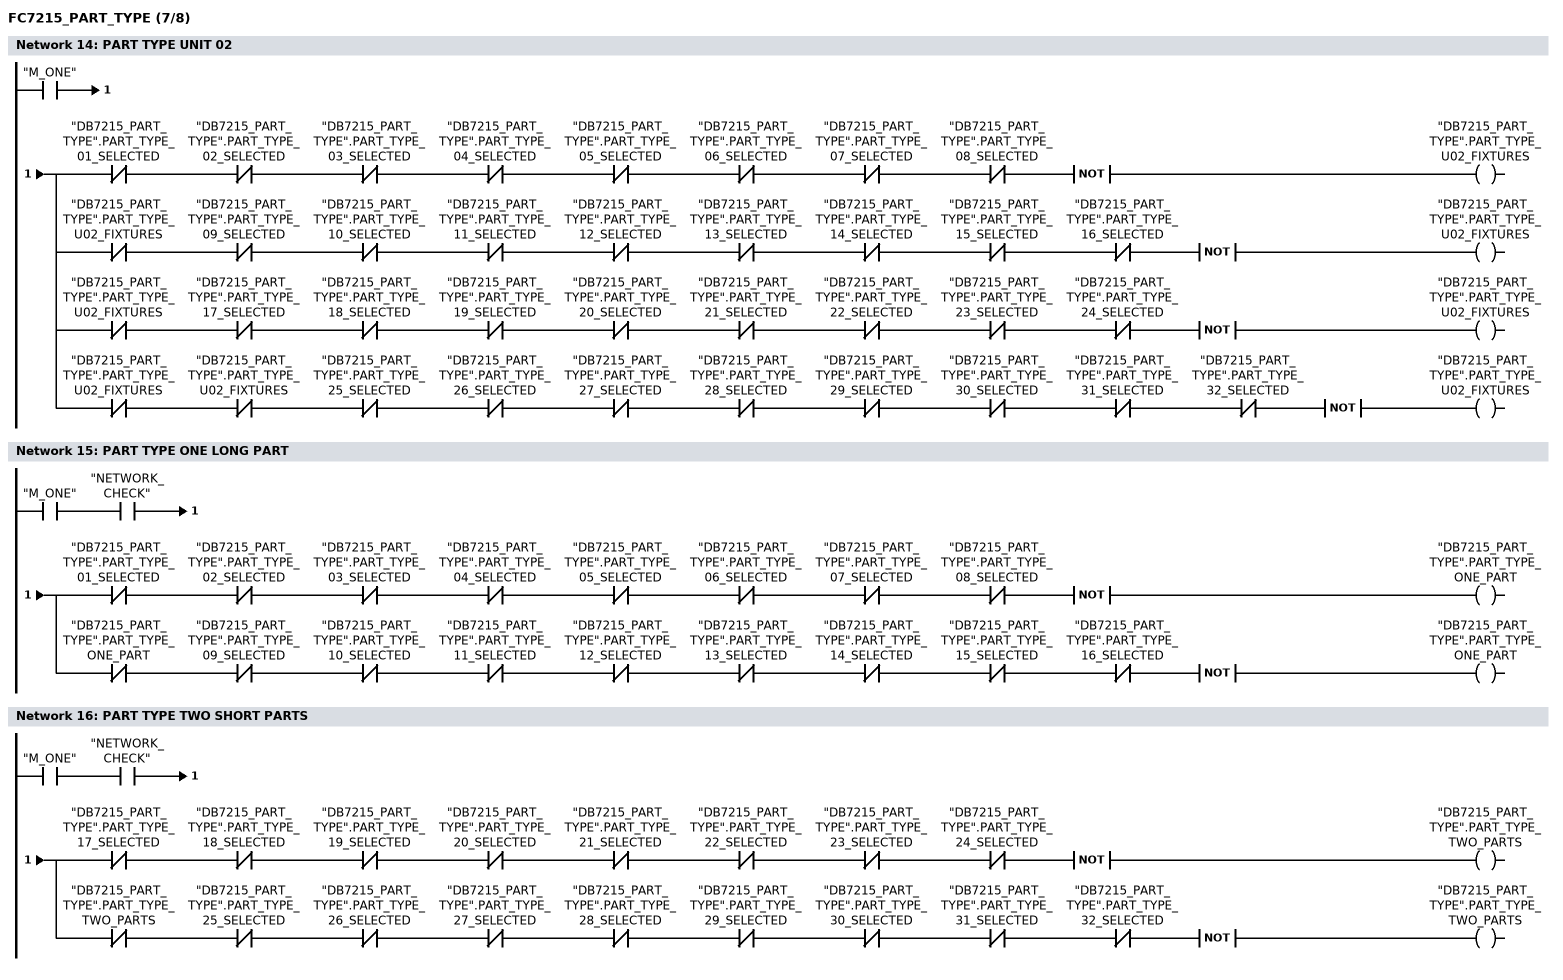
   RUNG wire#powerrail
      Contact( "M_ONE" )
      wire#w1
      I_Contact( "DB7215_PART_TYPE".PART_TYPE_01_SELECTED )
      I_Contact( "DB7215_PART_TYPE".PART_TYPE_02_SELECTED )
      I_Contact( "DB7215_PART_TYPE".PART_TYPE_03_SELECTED )
      I_Contact( "DB7215_PART_TYPE".PART_TYPE_04_SELECTED )
      I_Contact( "DB7215_PART_TYPE".PART_TYPE_05_SELECTED )
      I_Contact( "DB7215_PART_TYPE".PART_TYPE_06_SELECTED )
      I_Contact( "DB7215_PART_TYPE".PART_TYPE_07_SELECTED )
      I_Contact( "DB7215_PART_TYPE".PART_TYPE_08_SELECTED )
      Not()
      Coil( "DB7215_PART_TYPE".PART_TYPE_U02_FIXTURES )
   END_RUNG
   RUNG wire#w1
      I_Contact( "DB7215_PART_TYPE".PART_TYPE_U02_FIXTURES )
      I_Contact( "DB7215_PART_TYPE".PART_TYPE_09_SELECTED )
      I_Contact( "DB7215_PART_TYPE".PART_TYPE_10_SELECTED )
      I_Contact( "DB7215_PART_TYPE".PART_TYPE_11_SELECTED )
      I_Contact( "DB7215_PART_TYPE".PART_TYPE_12_SELECTED )
      I_Contact( "DB7215_PART_TYPE".PART_TYPE_13_SELECTED )
      I_Contact( "DB7215_PART_TYPE".PART_TYPE_14_SELECTED )
      I_Contact( "DB7215_PART_TYPE".PART_TYPE_15_SELECTED )
      I_Contact( "DB7215_PART_TYPE".PART_TYPE_16_SELECTED )
      Not()
      Coil( "DB7215_PART_TYPE".PART_TYPE_U02_FIXTURES )
   END_RUNG
   RUNG wire#w1
      I_Contact( "DB7215_PART_TYPE".PART_TYPE_U02_FIXTURES )
      I_Contact( "DB7215_PART_TYPE".PART_TYPE_17_SELECTED )
      I_Contact( "DB7215_PART_TYPE".PART_TYPE_18_SELECTED )
      I_Contact( "DB7215_PART_TYPE".PART_TYPE_19_SELECTED )
      I_Contact( "DB7215_PART_TYPE".PART_TYPE_20_SELECTED )
      I_Contact( "DB7215_PART_TYPE".PART_TYPE_21_SELECTED )
      I_Contact( "DB7215_PART_TYPE".PART_TYPE_22_SELECTED )
      I_Contact( "DB7215_PART_TYPE".PART_TYPE_23_SELECTED )
      I_Contact( "DB7215_PART_TYPE".PART_TYPE_24_SELECTED )
      Not()
      Coil( "DB7215_PART_TYPE".PART_TYPE_U02_FIXTURES )
   END_RUNG
   RUNG wire#w1
      I_Contact( "DB7215_PART_TYPE".PART_TYPE_U02_FIXTURES )
      I_Contact( "DB7215_PART_TYPE".PART_TYPE_U02_FIXTURES )
      I_Contact( "DB7215_PART_TYPE".PART_TYPE_25_SELECTED )
      I_Contact( "DB7215_PART_TYPE".PART_TYPE_26_SELECTED )
      I_Contact( "DB7215_PART_TYPE".PART_TYPE_27_SELECTED )
      I_Contact( "DB7215_PART_TYPE".PART_TYPE_28_SELECTED )
      I_Contact( "DB7215_PART_TYPE".PART_TYPE_29_SELECTED )
      I_Contact( "DB7215_PART_TYPE".PART_TYPE_30_SELECTED )
      I_Contact( "DB7215_PART_TYPE".PART_TYPE_31_SELECTED )
      I_Contact( "DB7215_PART_TYPE".PART_TYPE_32_SELECTED )
      Not()
      Coil( "DB7215_PART_TYPE".PART_TYPE_U02_FIXTURES )
   END_RUNG
   // the same network as SCL:
   "DB7215_PART_TYPE".PART_TYPE_U02_FIXTURES := NOT ("M_ONE" AND NOT "DB7215_PART_TYPE".PART_TYPE_01_SELECTED AND NOT "DB7215_PART_TYPE".PART_TYPE_02_SELECTED AND NOT "DB7215_PART_TYPE".PART_TYPE_03_SELECTED AND NOT "DB7215_PART_TYPE".PART_TYPE_04_SELECTED AND NOT "DB7215_PART_TYPE".PART_TYPE_05_SELECTED AND NOT "DB7215_PART_TYPE".PART_TYPE_06_SELECTED AND NOT "DB7215_PART_TYPE".PART_TYPE_07_SELECTED AND NOT "DB7215_PART_TYPE".PART_TYPE_08_SELECTED);
   "DB7215_PART_TYPE".PART_TYPE_U02_FIXTURES := NOT ("M_ONE" AND NOT "DB7215_PART_TYPE".PART_TYPE_U02_FIXTURES AND NOT "DB7215_PART_TYPE".PART_TYPE_09_SELECTED AND NOT "DB7215_PART_TYPE".PART_TYPE_10_SELECTED AND NOT "DB7215_PART_TYPE".PART_TYPE_11_SELECTED AND NOT "DB7215_PART_TYPE".PART_TYPE_12_SELECTED AND NOT "DB7215_PART_TYPE".PART_TYPE_13_SELECTED AND NOT "DB7215_PART_TYPE".PART_TYPE_14_SELECTED AND NOT "DB7215_PART_TYPE".PART_TYPE_15_SELECTED AND NOT "DB7215_PART_TYPE".PART_TYPE_16_SELECTED);
   "DB7215_PART_TYPE".PART_TYPE_U02_FIXTURES := NOT ("M_ONE" AND NOT "DB7215_PART_TYPE".PART_TYPE_U02_FIXTURES AND NOT "DB7215_PART_TYPE".PART_TYPE_17_SELECTED AND NOT "DB7215_PART_TYPE".PART_TYPE_18_SELECTED AND NOT "DB7215_PART_TYPE".PART_TYPE_19_SELECTED AND NOT "DB7215_PART_TYPE".PART_TYPE_20_SELECTED AND NOT "DB7215_PART_TYPE".PART_TYPE_21_SELECTED AND NOT "DB7215_PART_TYPE".PART_TYPE_22_SELECTED AND NOT "DB7215_PART_TYPE".PART_TYPE_23_SELECTED AND NOT "DB7215_PART_TYPE".PART_TYPE_24_SELECTED);
   "DB7215_PART_TYPE".PART_TYPE_U02_FIXTURES := NOT ("M_ONE" AND NOT "DB7215_PART_TYPE".PART_TYPE_U02_FIXTURES AND NOT "DB7215_PART_TYPE".PART_TYPE_U02_FIXTURES AND NOT "DB7215_PART_TYPE".PART_TYPE_25_SELECTED AND NOT "DB7215_PART_TYPE".PART_TYPE_26_SELECTED AND NOT "DB7215_PART_TYPE".PART_TYPE_27_SELECTED AND NOT "DB7215_PART_TYPE".PART_TYPE_28_SELECTED AND NOT "DB7215_PART_TYPE".PART_TYPE_29_SELECTED AND NOT "DB7215_PART_TYPE".PART_TYPE_30_SELECTED AND NOT "DB7215_PART_TYPE".PART_TYPE_31_SELECTED AND NOT "DB7215_PART_TYPE".PART_TYPE_32_SELECTED);
END_REGION

REGION Network 15: PART TYPE ONE LONG PART
   RUNG wire#powerrail
      Contact( "M_ONE" )
      Contact( "NETWORK_CHECK" )
      wire#w1
      I_Contact( "DB7215_PART_TYPE".PART_TYPE_01_SELECTED )
      I_Contact( "DB7215_PART_TYPE".PART_TYPE_02_SELECTED )
      I_Contact( "DB7215_PART_TYPE".PART_TYPE_03_SELECTED )
      I_Contact( "DB7215_PART_TYPE".PART_TYPE_04_SELECTED )
      I_Contact( "DB7215_PART_TYPE".PART_TYPE_05_SELECTED )
      I_Contact( "DB7215_PART_TYPE".PART_TYPE_06_SELECTED )
      I_Contact( "DB7215_PART_TYPE".PART_TYPE_07_SELECTED )
      I_Contact( "DB7215_PART_TYPE".PART_TYPE_08_SELECTED )
      Not()
      Coil( "DB7215_PART_TYPE".PART_TYPE_ONE_PART )
   END_RUNG
   RUNG wire#w1
      I_Contact( "DB7215_PART_TYPE".PART_TYPE_ONE_PART )
      I_Contact( "DB7215_PART_TYPE".PART_TYPE_09_SELECTED )
      I_Contact( "DB7215_PART_TYPE".PART_TYPE_10_SELECTED )
      I_Contact( "DB7215_PART_TYPE".PART_TYPE_11_SELECTED )
      I_Contact( "DB7215_PART_TYPE".PART_TYPE_12_SELECTED )
      I_Contact( "DB7215_PART_TYPE".PART_TYPE_13_SELECTED )
      I_Contact( "DB7215_PART_TYPE".PART_TYPE_14_SELECTED )
      I_Contact( "DB7215_PART_TYPE".PART_TYPE_15_SELECTED )
      I_Contact( "DB7215_PART_TYPE".PART_TYPE_16_SELECTED )
      Not()
      Coil( "DB7215_PART_TYPE".PART_TYPE_ONE_PART )
   END_RUNG
   // the same network as SCL:
   #_w1 := "M_ONE" AND "NETWORK_CHECK";
   "DB7215_PART_TYPE".PART_TYPE_ONE_PART := NOT (#_w1 AND NOT "DB7215_PART_TYPE".PART_TYPE_01_SELECTED AND NOT "DB7215_PART_TYPE".PART_TYPE_02_SELECTED AND NOT "DB7215_PART_TYPE".PART_TYPE_03_SELECTED AND NOT "DB7215_PART_TYPE".PART_TYPE_04_SELECTED AND NOT "DB7215_PART_TYPE".PART_TYPE_05_SELECTED AND NOT "DB7215_PART_TYPE".PART_TYPE_06_SELECTED AND NOT "DB7215_PART_TYPE".PART_TYPE_07_SELECTED AND NOT "DB7215_PART_TYPE".PART_TYPE_08_SELECTED);
   "DB7215_PART_TYPE".PART_TYPE_ONE_PART := NOT (#_w1 AND NOT "DB7215_PART_TYPE".PART_TYPE_ONE_PART AND NOT "DB7215_PART_TYPE".PART_TYPE_09_SELECTED AND NOT "DB7215_PART_TYPE".PART_TYPE_10_SELECTED AND NOT "DB7215_PART_TYPE".PART_TYPE_11_SELECTED AND NOT "DB7215_PART_TYPE".PART_TYPE_12_SELECTED AND NOT "DB7215_PART_TYPE".PART_TYPE_13_SELECTED AND NOT "DB7215_PART_TYPE".PART_TYPE_14_SELECTED AND NOT "DB7215_PART_TYPE".PART_TYPE_15_SELECTED AND NOT "DB7215_PART_TYPE".PART_TYPE_16_SELECTED);
END_REGION

REGION Network 16: PART TYPE TWO SHORT PARTS
   RUNG wire#powerrail
      Contact( "M_ONE" )
      Contact( "NETWORK_CHECK" )
      wire#w1
      I_Contact( "DB7215_PART_TYPE".PART_TYPE_17_SELECTED )
      I_Contact( "DB7215_PART_TYPE".PART_TYPE_18_SELECTED )
      I_Contact( "DB7215_PART_TYPE".PART_TYPE_19_SELECTED )
      I_Contact( "DB7215_PART_TYPE".PART_TYPE_20_SELECTED )
      I_Contact( "DB7215_PART_TYPE".PART_TYPE_21_SELECTED )
      I_Contact( "DB7215_PART_TYPE".PART_TYPE_22_SELECTED )
      I_Contact( "DB7215_PART_TYPE".PART_TYPE_23_SELECTED )
      I_Contact( "DB7215_PART_TYPE".PART_TYPE_24_SELECTED )
      Not()
      Coil( "DB7215_PART_TYPE".PART_TYPE_TWO_PARTS )
   END_RUNG
   RUNG wire#w1
      I_Contact( "DB7215_PART_TYPE".PART_TYPE_TWO_PARTS )
      I_Contact( "DB7215_PART_TYPE".PART_TYPE_25_SELECTED )
      I_Contact( "DB7215_PART_TYPE".PART_TYPE_26_SELECTED )
      I_Contact( "DB7215_PART_TYPE".PART_TYPE_27_SELECTED )
      I_Contact( "DB7215_PART_TYPE".PART_TYPE_28_SELECTED )
      I_Contact( "DB7215_PART_TYPE".PART_TYPE_29_SELECTED )
      I_Contact( "DB7215_PART_TYPE".PART_TYPE_30_SELECTED )
      I_Contact( "DB7215_PART_TYPE".PART_TYPE_31_SELECTED )
      I_Contact( "DB7215_PART_TYPE".PART_TYPE_32_SELECTED )
      Not()
      Coil( "DB7215_PART_TYPE".PART_TYPE_TWO_PARTS )
   END_RUNG
   // the same network as SCL:
   #_w1 := "M_ONE" AND "NETWORK_CHECK";
   "DB7215_PART_TYPE".PART_TYPE_TWO_PARTS := NOT (#_w1 AND NOT "DB7215_PART_TYPE".PART_TYPE_17_SELECTED AND NOT "DB7215_PART_TYPE".PART_TYPE_18_SELECTED AND NOT "DB7215_PART_TYPE".PART_TYPE_19_SELECTED AND NOT "DB7215_PART_TYPE".PART_TYPE_20_SELECTED AND NOT "DB7215_PART_TYPE".PART_TYPE_21_SELECTED AND NOT "DB7215_PART_TYPE".PART_TYPE_22_SELECTED AND NOT "DB7215_PART_TYPE".PART_TYPE_23_SELECTED AND NOT "DB7215_PART_TYPE".PART_TYPE_24_SELECTED);
   "DB7215_PART_TYPE".PART_TYPE_TWO_PARTS := NOT (#_w1 AND NOT "DB7215_PART_TYPE".PART_TYPE_TWO_PARTS AND NOT "DB7215_PART_TYPE".PART_TYPE_25_SELECTED AND NOT "DB7215_PART_TYPE".PART_TYPE_26_SELECTED AND NOT "DB7215_PART_TYPE".PART_TYPE_27_SELECTED AND NOT "DB7215_PART_TYPE".PART_TYPE_28_SELECTED AND NOT "DB7215_PART_TYPE".PART_TYPE_29_SELECTED AND NOT "DB7215_PART_TYPE".PART_TYPE_30_SELECTED AND NOT "DB7215_PART_TYPE".PART_TYPE_31_SELECTED AND NOT "DB7215_PART_TYPE".PART_TYPE_32_SELECTED);
END_REGION

REGION Network 17: PART TYPE SELECTED FAULT
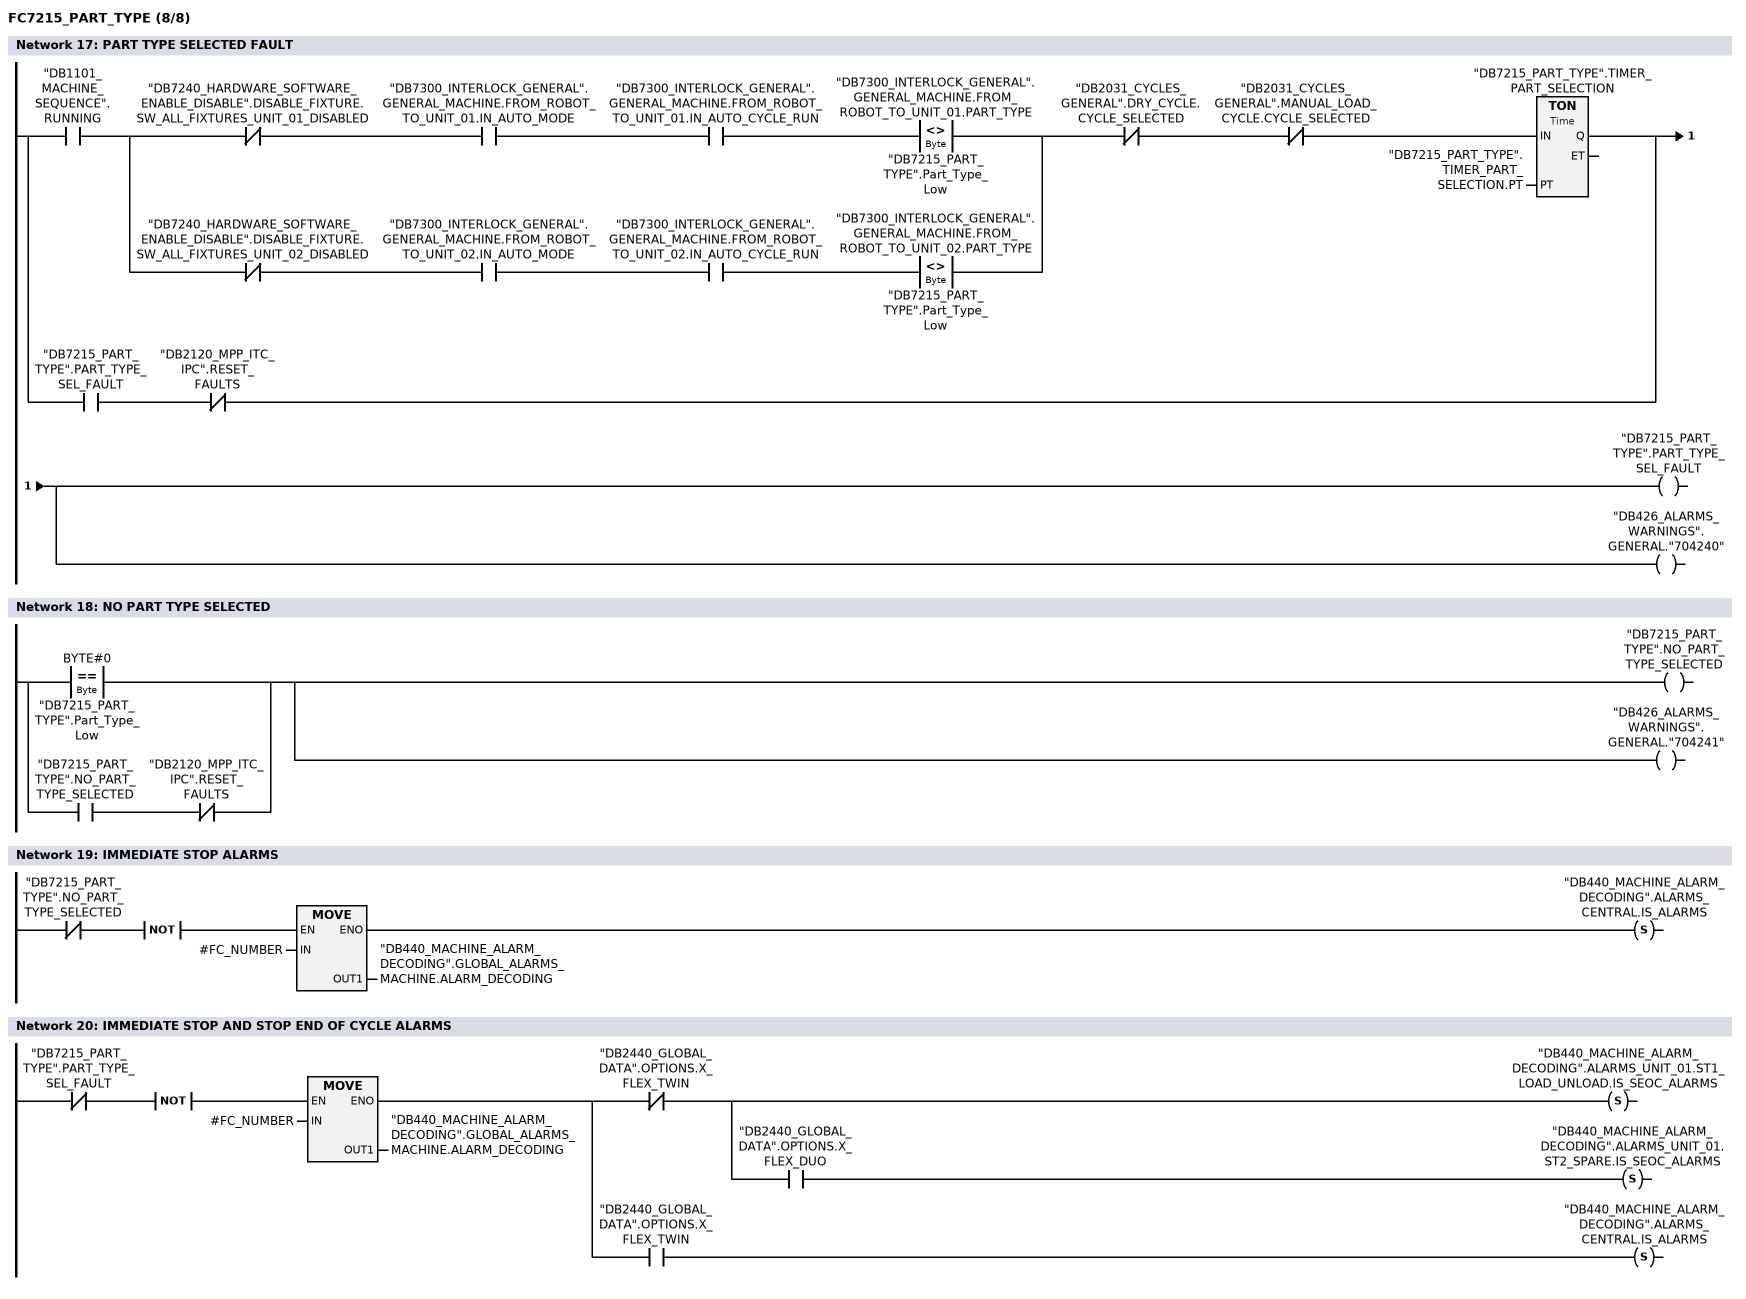
   RUNG wire#powerrail
      Contact( "DB1101_MACHINE_SEQUENCE".RUNNING )
      wire#w1
      I_Contact( "DB7240_HARDWARE_SOFTWARE_ENABLE_DISABLE".DISABLE_FIXTURE.SW_ALL_FIXTURES_UNIT_01_DISABLED )
      Contact( "DB7300_INTERLOCK_GENERAL".GENERAL_MACHINE.FROM_ROBOT_TO_UNIT_01.IN_AUTO_MODE )
      Contact( "DB7300_INTERLOCK_GENERAL".GENERAL_MACHINE.FROM_ROBOT_TO_UNIT_01.IN_AUTO_CYCLE_RUN )
      { S7_Templates := "SrcType := Byte" } NE_Contact(in1 := "DB7300_INTERLOCK_GENERAL".GENERAL_MACHINE.FROM_ROBOT_TO_UNIT_01.PART_TYPE, in2 := "DB7215_PART_TYPE".Part_Type_Low)
      wire#w2
      I_Contact( "DB2031_CYCLES_GENERAL".DRY_CYCLE.CYCLE_SELECTED )
      I_Contact( "DB2031_CYCLES_GENERAL".MANUAL_LOAD_CYCLE.CYCLE_SELECTED )
      { S7_Templates := "time_type := Time" } "DB7215_PART_TYPE".TIMER_PART_SELECTION.TON(pt := "DB7215_PART_TYPE".TIMER_PART_SELECTION.PT, et =>)
      wire#w3
      Coil( "DB7215_PART_TYPE".PART_TYPE_SEL_FAULT )
   END_RUNG
   RUNG wire#w1
      I_Contact( "DB7240_HARDWARE_SOFTWARE_ENABLE_DISABLE".DISABLE_FIXTURE.SW_ALL_FIXTURES_UNIT_02_DISABLED )
      Contact( "DB7300_INTERLOCK_GENERAL".GENERAL_MACHINE.FROM_ROBOT_TO_UNIT_02.IN_AUTO_MODE )
      Contact( "DB7300_INTERLOCK_GENERAL".GENERAL_MACHINE.FROM_ROBOT_TO_UNIT_02.IN_AUTO_CYCLE_RUN )
      { S7_Templates := "SrcType := Byte" } NE_Contact(in1 := "DB7300_INTERLOCK_GENERAL".GENERAL_MACHINE.FROM_ROBOT_TO_UNIT_02.PART_TYPE, in2 := "DB7215_PART_TYPE".Part_Type_Low)
   END_RUNG wire#w2
   RUNG wire#powerrail
      Contact( "DB7215_PART_TYPE".PART_TYPE_SEL_FAULT )
      I_Contact( "DB2120_MPP_ITC_IPC".RESET_FAULTS )
   END_RUNG wire#w3
   RUNG wire#w3
      Coil( "DB426_ALARMS_WARNINGS".GENERAL."704240" )
   END_RUNG
   // the same network as SCL:
   "DB7215_PART_TYPE".TIMER_PART_SELECTION.TON(IN := "DB1101_MACHINE_SEQUENCE".RUNNING AND ((NOT "DB7240_HARDWARE_SOFTWARE_ENABLE_DISABLE".DISABLE_FIXTURE.SW_ALL_FIXTURES_UNIT_01_DISABLED AND "DB7300_INTERLOCK_GENERAL".GENERAL_MACHINE.FROM_ROBOT_TO_UNIT_01.IN_AUTO_MODE AND "DB7300_INTERLOCK_GENERAL".GENERAL_MACHINE.FROM_ROBOT_TO_UNIT_01.IN_AUTO_CYCLE_RUN AND ("DB7300_INTERLOCK_GENERAL".GENERAL_MACHINE.FROM_ROBOT_TO_UNIT_01.PART_TYPE <> "DB7215_PART_TYPE".Part_Type_Low)) OR (NOT "DB7240_HARDWARE_SOFTWARE_ENABLE_DISABLE".DISABLE_FIXTURE.SW_ALL_FIXTURES_UNIT_02_DISABLED AND "DB7300_INTERLOCK_GENERAL".GENERAL_MACHINE.FROM_ROBOT_TO_UNIT_02.IN_AUTO_MODE AND "DB7300_INTERLOCK_GENERAL".GENERAL_MACHINE.FROM_ROBOT_TO_UNIT_02.IN_AUTO_CYCLE_RUN AND ("DB7300_INTERLOCK_GENERAL".GENERAL_MACHINE.FROM_ROBOT_TO_UNIT_02.PART_TYPE <> "DB7215_PART_TYPE".Part_Type_Low))) AND NOT "DB2031_CYCLES_GENERAL".DRY_CYCLE.CYCLE_SELECTED AND NOT "DB2031_CYCLES_GENERAL".MANUAL_LOAD_CYCLE.CYCLE_SELECTED,
                           PT := "DB7215_PART_TYPE".TIMER_PART_SELECTION.PT);
   "DB7215_PART_TYPE".PART_TYPE_SEL_FAULT := "DB7215_PART_TYPE".TIMER_PART_SELECTION.Q OR ("DB7215_PART_TYPE".PART_TYPE_SEL_FAULT AND NOT "DB2120_MPP_ITC_IPC".RESET_FAULTS);
   "DB426_ALARMS_WARNINGS".GENERAL."704240" := "DB7215_PART_TYPE".PART_TYPE_SEL_FAULT;
END_REGION

REGION Network 18: NO PART TYPE SELECTED
   RUNG wire#powerrail
      { S7_Templates := "SrcType := Byte" } EQ_Contact(in1 := BYTE#0, in2 := "DB7215_PART_TYPE".Part_Type_Low)
      wire#w1
      Coil( "DB7215_PART_TYPE".NO_PART_TYPE_SELECTED )
   END_RUNG
   RUNG wire#powerrail
      Contact( "DB7215_PART_TYPE".NO_PART_TYPE_SELECTED )
      I_Contact( "DB2120_MPP_ITC_IPC".RESET_FAULTS )
   END_RUNG wire#w1
   RUNG wire#w1
      Coil( "DB426_ALARMS_WARNINGS".GENERAL."704241" )
   END_RUNG
   // the same network as SCL:
   "DB7215_PART_TYPE".NO_PART_TYPE_SELECTED := (BYTE#0 = "DB7215_PART_TYPE".Part_Type_Low) OR ("DB7215_PART_TYPE".NO_PART_TYPE_SELECTED AND NOT "DB2120_MPP_ITC_IPC".RESET_FAULTS);
   "DB426_ALARMS_WARNINGS".GENERAL."704241" := "DB7215_PART_TYPE".NO_PART_TYPE_SELECTED;
END_REGION

REGION Network 19: IMMEDIATE STOP ALARMS
   RUNG wire#powerrail
      I_Contact( "DB7215_PART_TYPE".NO_PART_TYPE_SELECTED )
      Not()
      { S7_GenerateENO := "TRUE" } Move(in := #FC_NUMBER, out1 => "DB440_MACHINE_ALARM_DECODING".GLOBAL_ALARMS_MACHINE.ALARM_DECODING)
      S_Coil( "DB440_MACHINE_ALARM_DECODING".ALARMS_CENTRAL.IS_ALARMS )
   END_RUNG
   // the same network as SCL:
   // ENO of a box is taken as its EN; it also drops when the box reports an error
   IF NOT (NOT "DB7215_PART_TYPE".NO_PART_TYPE_SELECTED) THEN
       "DB440_MACHINE_ALARM_DECODING".GLOBAL_ALARMS_MACHINE.ALARM_DECODING := #FC_NUMBER;
       "DB440_MACHINE_ALARM_DECODING".ALARMS_CENTRAL.IS_ALARMS := TRUE;
   END_IF;
END_REGION

REGION Network 20: IMMEDIATE STOP AND STOP END OF CYCLE ALARMS
   RUNG wire#powerrail
      I_Contact( "DB7215_PART_TYPE".PART_TYPE_SEL_FAULT )
      Not()
      { S7_GenerateENO := "TRUE" } Move(in := #FC_NUMBER, out1 => "DB440_MACHINE_ALARM_DECODING".GLOBAL_ALARMS_MACHINE.ALARM_DECODING)
      wire#w1
      I_Contact( "DB2440_GLOBAL_DATA".OPTIONS.X_FLEX_TWIN )
      wire#w2
      S_Coil( "DB440_MACHINE_ALARM_DECODING".ALARMS_UNIT_01.ST1_LOAD_UNLOAD.IS_SEOC_ALARMS )
   END_RUNG
   RUNG wire#w2
      Contact( "DB2440_GLOBAL_DATA".OPTIONS.X_FLEX_DUO )
      S_Coil( "DB440_MACHINE_ALARM_DECODING".ALARMS_UNIT_01.ST2_SPARE.IS_SEOC_ALARMS )
   END_RUNG
   RUNG wire#w1
      Contact( "DB2440_GLOBAL_DATA".OPTIONS.X_FLEX_TWIN )
      S_Coil( "DB440_MACHINE_ALARM_DECODING".ALARMS_CENTRAL.IS_ALARMS )
   END_RUNG
   // the same network as SCL:
   // ENO of a box is taken as its EN; it also drops when the box reports an error
   #_w1 := NOT (NOT "DB7215_PART_TYPE".PART_TYPE_SEL_FAULT);
   IF #_w1 THEN "DB440_MACHINE_ALARM_DECODING".GLOBAL_ALARMS_MACHINE.ALARM_DECODING := #FC_NUMBER; END_IF;
   #_w2 := #_w1 AND NOT "DB2440_GLOBAL_DATA".OPTIONS.X_FLEX_TWIN;
   IF #_w2 THEN "DB440_MACHINE_ALARM_DECODING".ALARMS_UNIT_01.ST1_LOAD_UNLOAD.IS_SEOC_ALARMS := TRUE; END_IF;
   IF #_w2 AND "DB2440_GLOBAL_DATA".OPTIONS.X_FLEX_DUO THEN
       "DB440_MACHINE_ALARM_DECODING".ALARMS_UNIT_01.ST2_SPARE.IS_SEOC_ALARMS := TRUE;
   END_IF;
   IF #_w1 AND "DB2440_GLOBAL_DATA".OPTIONS.X_FLEX_TWIN THEN
       "DB440_MACHINE_ALARM_DECODING".ALARMS_CENTRAL.IS_ALARMS := TRUE;
   END_IF;
END_REGION
END_FUNCTION
